TYPE ST_IOOutput :
STRUCT
	QxLampeRouge AT%Q*:BOOL;
	QxLampeVerte AT%Q* : BOOL;
	QxLampeOrange AT%Q* :BOOL;
END_STRUCT
END_TYPE

(* stored: Version 1.1.0.1, ProductVersion 3.1.4020.6
   DUT ST_IOOutput: Id {b700e6de-0ef7-4bf2-abff-1f65fee3d439} *)
